PROGRAM _Discharge
VAR_INPUT
	i_bStart					:BOOL;
	i_bStartSieve				:BOOL;
	i_bStopSieve				:BOOL;
	i_bStartMixer				:BOOL;
	i_bStopMixer				:BOOL;
	i_iPhaseEndpoint			:INT;
	i_stDsichargeTime			:ST_HMI_Time;
	i_bBarrelInPosition			:BOOL;
	i_bConfirmFinishPhase		:BOOL;
	i_rMixerSpeed				:REAL;
	i_rSieveSpeed				:REAL;
END_VAR
VAR
	Seq_Time					:ARRAY[0..9] OF TIME;
	bSieveStop					:BOOL;
	bMixerStop					:BOOL;
	tonDelayPrompt				:TON;
END_VAR
VAR_OUTPUT
	q_stCmd						:ST_ProcessCmd;
	q_bRunning					:BOOL;
	q_bFinished					:BOOL;
	q_bPromptReq				:BOOL;
	q_tStepTime					:TIME;
	
END_VAR
VAR PERSISTENT
	iStep						:INT;
	iPrevStep					:INT;
	Seq_TON						:ARRAY[0..9] OF FB_TONP;
	tonStepTime					:FB_TONP;
	stSeqControl				:ST_SeqControl;
END_VAR

//****************RECIPE CALCULATIONS*********************
Seq_Time[1]:=DINT_TO_TIME(i_stDsichargeTime.mins)*60000 + 
			 DINT_TO_TIME(i_stDsichargeTime.sec)*1000;

//****************SEQUENE STATE AND CONTROL*********************
q_bRunning:=iStep<>0;
//Finish sequence if phase change is requested
IF q_bRunning AND (GV.stControl.bNext OR GV.stControl.bPrevious OR GV.stControl.bJump) THEN
	iStep:=1000;
END_IF
//Idle if phase is not active
IF NOT i_bStart THEN
	iStep:=0;
END_IF

//Timers
Seq_TON[1](IN:=(iStep=500), PAUSE:=GV.stControl.bPaused, PT:=Seq_Time[1]);

tonDelayPrompt(IN:=(iStep=500),PT:=T#30S);
//****************SEQUENCE*********************
CASE iStep OF
	0:
	IF i_bStart THEN
		q_bFinished := FALSE;
		iStep := 40;
	END_IF
	IF iStep <> 0 THEN
		iPrevStep:=0;
	END_IF
	
	40: //Barrel placed confirmation
	IF i_bBarrelInPosition THEN
		iStep:=50;
	END_IF
	IF iStep <> 40 THEN
		iPrevStep:=40;
	END_IF
	IF GV.stControl.bPaused THEN
		iStep := 40;
	END_IF
	
	50: //Check outlet
	IF IN.bOutletPos_Opened THEN
		iStep := 500;
	END_IF
	IF iStep <> 50 THEN
		iPrevStep:=50;
	END_IF
	IF GV.stControl.bPaused THEN
		iStep := 50;
	END_IF
	
	500://Wait for confirmation
	IF (i_iPhaseEndpoint = 0 AND Seq_TON[1].Q) OR 
	   (i_iPhaseEndpoint = 1 AND i_bConfirmFinishPhase) THEN
	   iStep:=1000;
	END_IF
	IF iStep <> 500 THEN
		iPrevStep := 500;
	END_IF
	IF GV.stControl.bPaused THEN
		iStep := 500;
	END_IF
	
	1000://Finish phase
	q_bFinished:=TRUE;
	IF GV.stControl.bPhaseFinished THEN
		q_bFinished:=FALSE;
		iStep:=0;
	END_IF
END_CASE

//****************COMMAND*********************
q_bPromptReq:=(iStep=40) OR
			  (tonDelayPrompt.Q AND i_iPhaseEndpoint = 1);

//Outlet
IF F_StepCMP(iStep,50,0,0,0,0,0,0,0,0,0) THEN
	q_stCmd.bOutletClose:=FALSE;
	q_stCmd.bOutletOpen:=TRUE;
ELSE
	q_stCmd.bOutletClose:=FALSE;
	q_stCmd.bOutletOpen:=FALSE;
END_IF

//Mixer
IF i_bStartMixer THEN
	bMixerStop:=FALSE;
ELSIF i_bStopMixer THEN
	bMixerStop:=TRUE;
END_IF

IF F_StepCMP(iStep,500,0,0,0,0,0,0,0,0,0) AND IN.bOutletPos_Opened AND NOT bMixerStop THEN
	q_stCmd.bMixerStart:=TRUE;
	q_stCmd.rMixerSpeed:=i_rMixerSpeed;
ELSE
	q_stCmd.bMixerStart:=FALSE;
	q_stCmd.rMixerSpeed:=0;
END_IF

//Air valves
q_stCMd.bMixerAir:=F_StepCMP(iStep,500,0,0,0,0,0,0,0,0,0);

//Sieve
IF i_bStartSieve THEN
	bSieveStop:=FALSE;
ELSIF i_bStopSieve THEN
	bSieveStop:=TRUE;
END_IF

IF F_StepCMP(iStep,500,0,0,0,0,0,0,0,0,0) AND IN.bOutletPos_Opened AND NOT bSieveStop THEN
	q_stCmd.bSieveStart:=TRUE;
	q_stCmd.rSieveSpeed:=i_rSieveSpeed;
ELSE
	q_stCmd.bSieveStart:=FALSE;
	q_stCmd.rSieveSpeed:=0;
END_IF

//Statistic and Status
tonStepTime(IN:=q_bRunning OR MAIN.bFirstCycle,PAUSE:=GV.bUPSdetect,PT:=T#3H);
q_tStepTime:=tonStepTime.ET;

//Sequence control HMI
stSeqControl.iCurrentStep:=iStep;
stSeqControl.iPreviousStep:=iPrevStep;
stSeqControl.iRecipeType:=0;
stSeqControl.iPhaseType:=3;
stSeqControl.sPhaseTime:=F_TimerHMI(q_tStepTime);

stSeqControl.iStepNumbers[0]:=0;
stSeqControl.sStepDescription[0]:='Wait for phase start';

stSeqControl.iStepNumbers[1]:=40;
stSeqControl.sStepDescription[1]:='Wait confirmation for barrel in position';

stSeqControl.iStepNumbers[2]:=50;
stSeqControl.sStepDescription[2]:='Check if outlet is opened';

stSeqControl.iStepNumbers[3]:=500;
stSeqControl.sStepDescription[3]:='Discharging';

stSeqControl.iStepNumbers[4]:=1000;
stSeqControl.sStepDescription[4]:='Phase finished';

stSeqControl.iStepNumbers[5]:=0;
stSeqControl.sStepDescription[5]:='';

stSeqControl.iStepNumbers[6]:=0;
stSeqControl.sStepDescription[6]:='';

stSeqControl.iStepNumbers[7]:=0;
stSeqControl.sStepDescription[7]:='';

stSeqControl.iStepNumbers[8]:=0;
stSeqControl.sStepDescription[8]:='';

stSeqControl.iStepNumbers[9]:=0;
stSeqControl.sStepDescription[9]:='';

END_PROGRAM

(* stored: Version 1.1.0.1, ProductVersion 3.1.4024.12
   POU _Discharge: Id {34813e8e-0c54-45fa-b12b-607066094ebb}, SpecialFunc None *)
